// TIA Portal V18 export
// export: Created 2026-01-09T11:31:50.3546615Z, ExportSetting WithDefaults, DisplayName Totally Integrated Automation Portal, DisplayVersion V18 Update 5, DisplayName TIA Portal Openness, DisplayVersion V18 Update 5, DisplayName TIA Portal Teamcenter Gateway, DisplayVersion V18, DisplayName TIA Portal Version Control Interface, DisplayVersion V18, DisplayName SINAMICS Startdrive Advanced, DisplayVersion V18 SP2 Update 1, DisplayName SINAMICS Startdrive G110M, G120, G120C, G120D, G120P, G115D, DisplayVersion V18 SP2 Update 1, DisplayName SINAMICS Startdrive G130, G150, S120, S150, SINAMICS MV, S210, G220, S200, DisplayVersion V18 SP2 Update 1, DisplayName STEP 7 Professional, DisplayVersion V18 Update 5, DisplayName STEP 7 Safety, DisplayVersion V18, DisplayName WinCC Professional, DisplayVersion V18 Update 5
TagTable "过程数据"
  Status_FlowPart2 : Int  (PLC tag ST10_GeneralData.FlowPartStatus[2], CPU S71500-2PN_TP700, 1 s)
  Status_FlowPart1 : Int  (PLC tag ST10_GeneralData.FlowPartStatus[1], CPU S71500-2PN_TP700, 1 s)
  Status_FlowPart3 : Int  (PLC tag ST10_GeneralData.FlowPartStatus[3], CPU S71500-2PN_TP700, 1 s)
  Station1_PM_Num{3}_ProcessResult : DInt  (PLC tag ST10_PM.Num[3].ProcessResult, CPU S71500-2PN_TP700, 1 s)
